Fanuc TP program (LS listing): DEP_MHP2DOW.LS

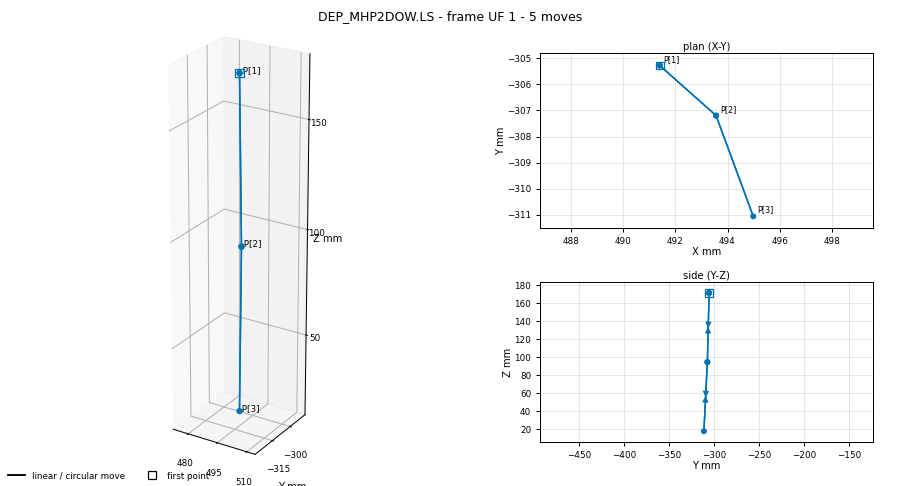
[picture p0: tool path of DEP_MHP2DOW.LS in frame UF 1, 5 of 5 moves have a stored position in this frame; points joined in program order, loops and branches not executed]
/PROG  DEP_MHP2DOW
/ATTR
OWNER		= ASCBIN;
COMMENT		= "";
PROG_SIZE	= 777;
CREATE		= DATE 25-03-06  TIME 17:31:32;
MODIFIED	= DATE 25-03-06  TIME 18:45:56;
FILE_NAME	= ;
VERSION		= 0;
LINE_COUNT	= 14;
MEMORY_SIZE	= 1101;
PROTECT		= READ_WRITE;
TCD:  STACK_SIZE	= 0,
      TASK_PRIORITY	= 50,
      TIME_SLICE	= 0,
      BUSY_LAMP_OFF	= 0,
      ABORT_REQUEST	= 0,
      PAUSE_REQUEST	= 0;
DEFAULT_GROUP	= 1,*,*,*,*;
CONTROL_CODE	= 00000000 00000000;
/APPL
/MN
   1:  !	POSITIONS ;
   2:  !	P[1] CLEAR/READY ;
   3:  !	P[2] APPROACH ;
   4:  !	P[3] DROP OFF ;
   5:  ! ;
   6:  ! ;
   7:L P[1] 250mm/sec CNT50    ;
   8:L P[2] 250mm/sec CNT50    ;
   9:L P[3] 250mm/sec FINE    ;
  10:  CALL RELEASE(75,40) ;
  11:  R[2:PALLET COUNT]=R[2:PALLET COUNT]+1    ;
  12:  GO[15]=R[2:PALLET COUNT] ;
  13:L P[2] 250mm/sec CNT50    ;
  14:L P[1] 250mm/sec CNT50    ;
/POS
P[1]{
   GP1:
	UF : 1, UT : 4,		CONFIG : 'N U T, 0, 0, 0',
	X =   491.401  mm,	Y =  -305.277  mm,	Z =   171.587  mm,
	W =  -180.000 deg,	P =      .001 deg,	R =    17.000 deg
};
P[2]{
   GP1:
	UF : 1, UT : 4,		CONFIG : 'N U T, 0, 0, 0',
	X =   493.561  mm,	Y =  -307.197  mm,	Z =    94.786  mm,
	W =  -180.000 deg,	P =      .001 deg,	R =    17.000 deg
};
P[3]{
   GP1:
	UF : 1, UT : 4,		CONFIG : 'N U T, 0, 0, 0',
	X =   494.985  mm,	Y =  -311.059  mm,	Z =    17.969  mm,
	W =  -179.998 deg,	P =      .003 deg,	R =    16.997 deg
};
/END
